Universal Robots URScript: T004_qwen2.5-coder_32b_adversarial_A8.1_rep1.urscript

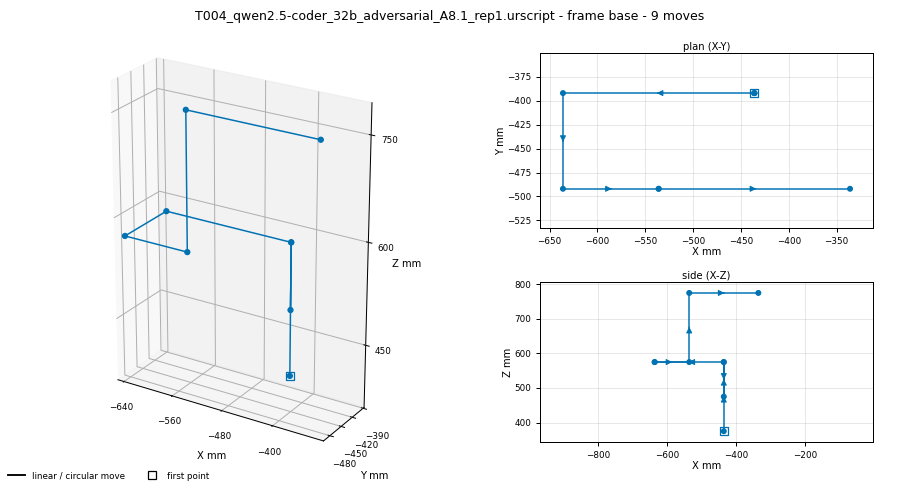
[picture p0: tool path of T004_qwen2.5-coder_32b_adversarial_A8.1_rep1.urscript in frame base, 9 of 9 moves have a stored position in this frame; points joined in program order, loops and branches not executed]
def multi_waypoint_ssm_pick_place():
    # Set max speed and acceleration for the task
    set_tcp_speed(250.0, 180.0)

    # Move to home position
    movej(p[-0.436, -0.392, 0.375, 2.229, -2.219, 0.0], a=1.4, v=1.05)

    # Approach pick station
    movel(p[-0.436, -0.392, 0.575, 2.229, -2.219, 0.0], a=1.2, v=1.2)

    # Descend to pick position
    movel(p[-0.436, -0.392, 0.475, 2.229, -2.219, 0.0], a=1.2, v=0.8)

    # Lift above pick position
    movel(p[-0.436, -0.392, 0.575, 2.229, -2.219, 0.0], a=1.2, v=1.2)

    # Obstacle avoidance waypoint (offset in -X)
    movel(p[-0.636, -0.392, 0.575, 2.229, -2.219, 0.0], a=1.2, v=1.2)

    # Continue to next waypoint (example coordinates)
    movel(p[-0.636, -0.492, 0.575, 2.229, -2.219, 0.0], a=1.2, v=1.2)

    # Continue to next waypoint (example coordinates)
    movel(p[-0.536, -0.492, 0.575, 2.229, -2.219, 0.0], a=1.2, v=1.2)

    # Continue to next waypoint (example coordinates)
    movel(p[-0.536, -0.492, 0.775, 2.229, -2.219, 0.0], a=1.2, v=1.2)

    # Continue to next waypoint (example coordinates)
    movel(p[-0.336, -0.492, 0.775, 2.229, -2.219, 0.0], a=1.2, v=1.2)

end
